PROGRAM MAIN
VAR
	SAVE_RETAIN: FB_S_UPS_CX51x0;
	puls_chiamata AT %I*: BOOL;
	sirena_canc AT %Q*: BOOL;
	apert_canc AT %Q*: BOOL;
	Sirena_cancello: TP;
	apertura_porta_ingr: TP;
	apert_canc1 : BOOL; //Apertura cancello per trasportatori
	apert_canc2 : BOOL; //Apertura cancello per dipendenti
	apert_canc3 : BOOL; //Apertura cancello con sensore e con allarme
	compr_pistone AT %Q* : BOOL;
	compr_vite AT %Q* : BOOL;
	luce : ARRAY [1..10] OF comando_luce;
	
	//controllo Energia
	energy_ch1_control AT %Q* : USINT;
	energy_ch2_control AT %Q* : USINT;
	energy_ch3_control AT %Q* : USINT;
	energy_ch1_dataIN AT %I* : INT;
	energy_ch2_dataIN AT %I* : INT;
	energy_ch3_dataIN AT %I* : INT;
	energy_ch1_state AT %I* : USINT;
	energy_ch2_state AT %I* : USINT;
	energy_ch3_state AT %I* : USINT;
	energy_function:INT;
	
	//Tempo_Cancello_trasp: RS;
	//Tempo_Cancello_Dip: RS;
	Entrata_Trasp: TP;
	timer_allarme: TON;
	Energydata_update: R_TRIG;
	alarm_counter: INT;
	Accensione_luci: F_TRIG;
	Spegnimento_luci: R_TRIG;
	Delay_allarme: TON;
	led_allarmeon: BOOL;
	ins_allarme: R_TRIG;
	ins_AUTOallarme: F_TRIG;
	allarme_off: R_TRIG;
	puls_allarme: TON;
	HMI_puls_allarme: TON; //Inserimento allarme da pannello
END_VAR

//ads_CX8080();
enocean();
DALI();
Ekey();
RISCALDAMENTO();
luci();
ULUX();
KNX();
Alarm();
// Salvataggio dati con UPS Interno
SAVE_RETAIN(
	sNetID:= '', 
	iPLCPort:= 851, 
	iUPSPort:= , 
	tTimeout:= , 
	eUpsMode:= , 
	ePersistentMode:= , 
	tRecoverTime:= , 
	bPowerFailDetect=> , 
	eState=> );

(*Gestione e Conversione ORA*)
time_now := (ORA_PLC.TIMESTR.wHour*100)+ ora_plc.TIMESTR.wMinute;
(*Gestione Orari GUEST*)
GuestIN_OK:= ((time_now>=time_work_IN1 AND time_now<=time_work_OUT1)
			OR (time_now>=time_work_IN2 AND time_now<=time_work_OUT2))
			AND allarme_Attivo=0;
(*Gestione Orari USER*)
IF holidays OR ora_plc.TIMESTR.wDayOfWeek=0 THEN
	USERIN_OK:=FALSE;
ELSIF (ora_plc.TIMESTR.wDayOfWeek=6 AND saturday_work) AND (time_now>=time_IN1 AND time_now<=time_OUT1) THEN
	USERIN_OK:=TRUE;
ELSIF (ora_plc.TIMESTR.wDayOfWeek>=1 AND ora_plc.TIMESTR.wDayOfWeek<=5) AND ((time_now>=time_IN1 AND time_now<=time_OUT1)
																		OR (time_now>=time_IN2 AND time_now<=time_OUT2)) THEN
	USERIN_OK:=TRUE;
ELSE
	USERIN_OK:=FALSE;	
END_IF
(*Segnale allarme*)
(*allarme_off(CLK:= time_now=0730, Q=> );
IF allarme_off.Q THEN
	allarme:=FALSE;
END_IF*)
//Inserimento allarme con pulsante a muro o HMI
puls_allarme(IN:= puld1, PT:= T#5S, Q=> , ET=> );
HMI_puls_allarme(IN:= HMI_Allarme, PT:= T#5S, Q=> , ET=> );
IF puls_allarme.Q OR hmi_puls_allarme.Q THEN
	allarme_Attivo:=1;
END_IF
ins_allarme(CLK:= time_now=1730, Q=> );
ins_AUTOallarme(CLK:= time_now=1730, Q=> );
IF ins_allarme.Q AND auto_allarm THEN
	allarme_Attivo:=1;
END_IF
IF ins_AUTOallarme.Q THEN
	auto_allarm:=TRUE;
END_IF
luce[1].pulsante:=TRUE;
//Compressori
compr_vite:=TRUE;
compr_pistone:=allarme_Attivo=0;

//--> GESTIONE CANCELLO
//Apertura cancello per tipo utente per dipendenti + spegnimento allarme
IF ekey_scanner_cancello.bGoodFinger AND utenti[ekey_scanner_cancello.byRecUserID].user_type=3 THEN
	apert_canc2:=TRUE;
	allarme_attivo:=0;
ELSIF ekey_scanner_cancello.bGoodFinger AND utenti[ekey_scanner_cancello.byRecUserID].user_type=0 AND userin_OK THEN
	apert_canc2:=TRUE;
	allarme_Attivo:=0;
ELSE
	apert_canc2:=FALSE;
END_IF
//Spegnimento allarme con scanner ingresso
IF ekey_scanner_ingresso.bGoodFinger AND utenti[ekey_scanner_cancello.byRecUserID].user_type=3 THEN
	allarme_Attivo:=0;
END_IF
//Spegnimento allarme automatico con scanner ingresso per pulizia
IF ekey_scanner_ingresso.bGoodFinger AND ekey_scanner_ingresso.byRecUserID=26 AND allarme_Attivo=0 AND time_now<1730 THEN
	auto_allarm:=FALSE;
END_IF
//Apertura porta ingresso con ekey e HMI
apertura_porta_ingr(IN:= (ekey_scanner_ingresso.bGoodFinger AND allarme_Attivo=0) OR HMI_porta, PT:= T#1S, Q=> out_Pingresso, ET=> );
//Apertura cancello con pulsante per trasportatori
IF puls_chiamata AND guestin_ok THEN
	apert_canc1:=TRUE;
ELSE
	apert_canc1:=FALSE;
END_IF
//Apertura cancello con sensore auto e con allarme
timer_allarme(IN:= allarme_Attivo<>0, PT:= delay_allarme_on, Q=> , ET=> );
apert_canc3:=NOT timer_Allarme.Q AND sens_cancello_auto;

apert_canc:=apert_canc1 OR apert_canc2 OR apert_canc3 OR hmi_cancello OR IN_CITOR1;
Sirena_cancello(IN:= puls_chiamata, PT:= T#5S, Q=> sirena_canc, ET=> );

//Apertura cancello pedonale
OUT_Pcanc_ped:=IN_CITOR2 OR HMI_Cancelletto;
//<-- GESTIONE CANCELLO

//Controllo Energia	
CASE energy_function OF
	0:	energy_ch1_control :=0;
		IF energy_ch1_control=energy_ch1_state THEN
			HMI_currentL1:=energy_ch1_dataIN;
			energy_function:=energy_function+1;
		END_IF;
	1:	energy_ch2_control :=0;
		IF energy_ch2_control=energy_ch2_state THEN
			HMI_currentL2:=energy_ch2_dataIN;
			energy_function:=energy_function+1;
		END_IF;
	2:	energy_ch3_control :=0;
		IF energy_ch3_control=energy_ch3_state THEN
			HMI_currentL3:=energy_ch3_dataIN;
			energy_function:=energy_function+1;
		END_IF;
	3:	energy_ch1_control :=1;
		IF energy_ch1_control=energy_ch1_state THEN
			HMI_voltageL1:=energy_ch1_dataIN;
			energy_function:=energy_function+1;
		END_IF;
	4:	energy_ch2_control :=1;
		IF energy_ch2_control=energy_ch2_state THEN
			HMI_voltageL2:=energy_ch2_dataIN;
			energy_function:=energy_function+1;
		END_IF;
	5:	energy_ch3_control :=1;
		IF energy_ch3_control=energy_ch3_state THEN
			HMI_voltageL3:=energy_ch3_dataIN;
			energy_function:=energy_function+1;
		END_IF;	
	6:	energy_ch1_control :=2;
		IF energy_ch1_control=energy_ch1_state THEN
			HMI_PowerL1:=energy_ch1_dataIN;
			energy_function:=energy_function+1;
		END_IF;
	7:	energy_ch2_control :=2;
		IF energy_ch2_control=energy_ch2_state THEN
			HMI_PowerL2:=energy_ch2_dataIN;
			energy_function:=energy_function+1;
		END_IF;
	8:	energy_ch3_control :=2;
		IF energy_ch3_control=energy_ch3_state THEN
			HMI_PowerL3:=energy_ch3_dataIN;
			energy_function:=energy_function+1;
		END_IF;	
	9:	energy_ch1_control :=4;
		IF energy_ch1_control=energy_ch1_state THEN
			HMI_energyL1:=energy_ch1_dataIN;
			energy_function:=energy_function+1;
		END_IF;
	10:	energy_ch2_control :=4;
		IF energy_ch2_control=energy_ch2_state THEN
			HMI_energyL2:=energy_ch2_dataIN;
			energy_function:=energy_function+1;
		END_IF;
	11:	energy_ch3_control :=4;
		IF energy_ch3_control=energy_ch3_state THEN
			HMI_energyL3:=energy_ch3_dataIN;
			energy_function:=energy_function+1;
		END_IF;	
	12:	energy_ch1_control :=8;
		IF energy_ch1_control=energy_ch1_state THEN
			HMI_frequencyL1:=energy_ch1_dataIN;
			energy_function:=energy_function+1;
		END_IF;
	13:	energy_ch2_control :=8;
		IF energy_ch2_control=energy_ch2_state THEN
			HMI_frequencyL2:=energy_ch2_dataIN;
			energy_function:=energy_function+1;
		END_IF;
	14:	energy_ch3_control :=8;
		IF energy_ch3_control=energy_ch3_state THEN
			HMI_frequencyL3:=energy_ch3_dataIN;
			energy_function:=0;
		END_IF;	
END_CASE;

ACTION ACT:
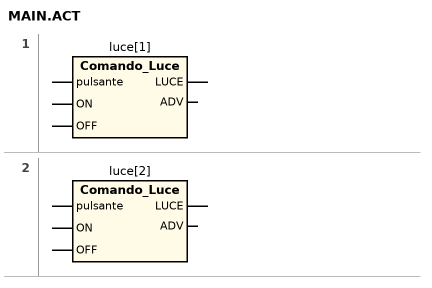
// NETWORK 1
luce[1](); // Comando_Luce

// NETWORK 2
luce[2](); // Comando_Luce
END_ACTION

END_PROGRAM

(* stored: Version 1.1.0.1, ProductVersion 3.1.4022.18
   POU MAIN: Id {e0859f41-33d8-4113-9dbe-37c16c52d498}, SpecialFunc None
   Action ACT: Id {85c3a37f-9c0f-43f9-9b74-f1aa6adfbeb0} *)
